FUNCTION FC_Error : STRING
VAR_INPUT
	eError : UDINT;
END_VAR
VAR
END_VAR

CASE eError OF
    // Global error codes
    16#00000000: FC_Error := 'No error';
    16#00000001: FC_Error := 'Internal error';
    16#00000002: FC_Error := 'No real time';
    16#00000003: FC_Error := 'Allocation locked – memory error';
    16#00000004: FC_Error := 'Mailbox full – ADS message could not be sent';
    16#00000005: FC_Error := 'Wrong HMSG';
    16#00000006: FC_Error := 'Target port not found – ADS server not started or reachable';
    16#00000007: FC_Error := 'Target computer not found – AMS route not found';
    16#00000008: FC_Error := 'Unknown command ID';
    16#00000009: FC_Error := 'Invalid task ID';
    16#0000000A: FC_Error := 'No IO';
    16#0000000B: FC_Error := 'Unknown AMS command';
    16#0000000C: FC_Error := 'Win32 error';
    16#0000000D: FC_Error := 'Port not connected';
    16#0000000E: FC_Error := 'Invalid AMS length';
    16#0000000F: FC_Error := 'Invalid AMS Net ID';
    16#00000010: FC_Error := 'Installation level too low – TwinCAT 2 license error';
    16#00000011: FC_Error := 'No debugging available';
    16#00000012: FC_Error := 'Port disabled – TwinCAT system service not started';
    16#00000013: FC_Error := 'Port already connected';
    16#00000014: FC_Error := 'AMS Sync Win32 error';
    16#00000015: FC_Error := 'AMS Sync timeout';
    16#00000016: FC_Error := 'AMS Sync error';
    16#00000017: FC_Error := 'No index map for AMS Sync';
    16#00000018: FC_Error := 'Invalid AMS port';
    16#00000019: FC_Error := 'No memory';
    16#0000001A: FC_Error := 'TCP send error';
    16#0000001B: FC_Error := 'Host unreachable';
    16#0000001C: FC_Error := 'Invalid AMS fragment';
    16#0000001D: FC_Error := 'TLS send error – secure ADS connection failed';
    16#0000001E: FC_Error := 'Access denied – secure ADS access denied';

    // Router error codes
    16#00000500: FC_Error := 'Locked memory cannot be allocated';
    16#00000501: FC_Error := 'Router memory size could not be changed';
    16#00000502: FC_Error := 'Mailbox reached maximum messages';
    16#00000503: FC_Error := 'Debug mailbox reached maximum messages';
    16#00000504: FC_Error := 'Unknown port type';
    16#00000505: FC_Error := 'Router not initialized';
    16#00000506: FC_Error := 'Port number already assigned';
    16#00000507: FC_Error := 'Port not registered';
    16#00000508: FC_Error := 'Maximum number of ports reached';
    16#00000509: FC_Error := 'Invalid port';
    16#0000050A: FC_Error := 'Router not active';
    16#0000050B: FC_Error := 'Mailbox reached maximum for fragmented messages';
    16#0000050C: FC_Error := 'Fragment timeout occurred';
    16#0000050D: FC_Error := 'Port removed';

    // General ADS error codes
    16#00000700: FC_Error := 'General device error';
    16#00000701: FC_Error := 'Service not supported by server';
    16#00000702: FC_Error := 'Invalid index group';
    16#00000703: FC_Error := 'Invalid index offset';
    16#00000704: FC_Error := 'Reading or writing not permitted';
    16#00000705: FC_Error := 'Parameter size not correct';
    16#00000706: FC_Error := 'Invalid data values';
    16#00000707: FC_Error := 'Device not ready';
    16#00000708: FC_Error := 'Device busy';
    16#00000709: FC_Error := 'Invalid operating system context';
    16#0000070A: FC_Error := 'Insufficient memory';
    16#0000070B: FC_Error := 'Invalid parameter values';
    16#0000070C: FC_Error := 'Not found (files, …)';
    16#0000070D: FC_Error := 'Syntax error in file or command';
    16#0000070E: FC_Error := 'Objects do not match';
    16#0000070F: FC_Error := 'Object already exists';
    16#00000710: FC_Error := 'Symbol not found';
    16#00000711: FC_Error := 'Invalid symbol version';
    16#00000712: FC_Error := 'Device in invalid state';
    16#00000713: FC_Error := 'AdsTransMode not supported';
    16#00000714: FC_Error := 'Notification handle invalid';
    16#00000715: FC_Error := 'Notification client not registered';
    16#00000716: FC_Error := 'No further handle available';
    16#00000717: FC_Error := 'Notification size too large';
    16#00000718: FC_Error := 'Device not initialized';
    16#00000719: FC_Error := 'Device timeout';
    16#0000071A: FC_Error := 'Interface query failed';
    16#0000071B: FC_Error := 'Wrong interface requested';
    16#0000071C: FC_Error := 'Class ID invalid';
    16#0000071D: FC_Error := 'Object ID invalid';
    16#0000071E: FC_Error := 'Request pending';
    16#0000071F: FC_Error := 'Request aborted';
    16#00000720: FC_Error := 'Signal warning';
    16#00000721: FC_Error := 'Invalid array index';
    16#00000722: FC_Error := 'Symbol not active';
    16#00000723: FC_Error := 'Access denied';
    16#00000724: FC_Error := 'License not found';
    16#00000725: FC_Error := 'License expired';
    16#00000726: FC_Error := 'License exceeded';
    16#00000727: FC_Error := 'Invalid license';
    16#00000728: FC_Error := 'System ID invalid';
    16#00000729: FC_Error := 'License not limited in time';
    16#0000072A: FC_Error := 'License time in future';
    16#0000072B: FC_Error := 'License period too long';
    16#0000072C: FC_Error := 'Exception at system startup';
    16#0000072D: FC_Error := 'License file read twice';
    16#0000072E: FC_Error := 'Invalid signature';
    16#0000072F: FC_Error := 'Invalid certificate';
    16#00000730: FC_Error := 'OEM public key not found';
    16#00000731: FC_Error := 'License not valid for system ID';
    16#00000732: FC_Error := 'Demo license prohibited';
    16#00000733: FC_Error := 'Invalid function ID';
    16#00000734: FC_Error := 'Value out of range';
    16#00000735: FC_Error := 'Invalid alignment';
    16#00000736: FC_Error := 'Invalid platform level';
    16#00000737: FC_Error := 'Forward to passive level';
    16#00000738: FC_Error := 'Forward to dispatch level';
    16#00000739: FC_Error := 'Forward to real-time';
    16#00000740: FC_Error := 'Client error';
    16#00000741: FC_Error := 'Service contains invalid parameter';
    16#00000742: FC_Error := 'Polling list empty';
    16#00000743: FC_Error := 'Var connection already in use';
    16#00000744: FC_Error := 'Called ID already in use';
    16#00000745: FC_Error := 'Timeout occurred';
    16#00000746: FC_Error := 'Win32 subsystem error';
    16#00000747: FC_Error := 'Invalid client timeout value';
    16#00000748: FC_Error := 'Port not open';
    16#00000749: FC_Error := 'No AMS address';
    16#00000750: FC_Error := 'Internal error in ADS sync';
    16#00000751: FC_Error := 'Hash table overflow';
    16#00000752: FC_Error := 'Key not found in table';
    16#00000753: FC_Error := 'No symbols in cache';
    16#00000754: FC_Error := 'Invalid response received';
    16#00000755: FC_Error := 'Sync port is locked';
    16#00000756: FC_Error := 'Request cancelled';
    // Additional General ADS error codes (added for completeness based on Beckhoff documentation)
    16#00000757: FC_Error := 'No real time';
    16#00000758: FC_Error := 'Real time extension not loaded';
    16#00000759: FC_Error := 'Real time extension not started';
    16#0000075A: FC_Error := 'Real time extension not configured';
    16#0000075B: FC_Error := 'Real time extension not initialized';
    16#0000075C: FC_Error := 'Real time extension not running';
    16#0000075D: FC_Error := 'Real time not supported on this CPU';
    16#0000075E: FC_Error := 'Real time not supported on this OS';
    16#0000075F: FC_Error := 'Real time extension error';
    16#00000760: FC_Error := 'Invalid driver version';
    16#00000761: FC_Error := 'Invalid driver handle';
    16#00000762: FC_Error := 'Driver not found';
    16#00000763: FC_Error := 'Driver not loaded';
    16#00000764: FC_Error := 'Driver not started';
    16#00000765: FC_Error := 'Driver not initialized';
    16#00000766: FC_Error := 'Driver not running';
    16#00000767: FC_Error := 'Driver error';
    16#00000768: FC_Error := 'Driver not supported';
    16#00000769: FC_Error := 'Driver already loaded';
    16#00000770: FC_Error := 'Invalid PLC project';
    16#00000771: FC_Error := 'PLC project not found';
    16#00000772: FC_Error := 'PLC project not loaded';
    16#00000773: FC_Error := 'PLC project not started';
    16#00000774: FC_Error := 'PLC project not running';
    16#00000775: FC_Error := 'PLC runtime error';
    16#00000780: FC_Error := 'Invalid route';
    16#00000781: FC_Error := 'Route not found';
    16#00000782: FC_Error := 'Route not active';
    16#00000783: FC_Error := 'Route not connected';
    16#00000784: FC_Error := 'Route timeout';
    16#00000785: FC_Error := 'Route error';
    16#00000790: FC_Error := 'Invalid AMS NetID';
    16#00000791: FC_Error := 'Invalid AMS port';
    16#00000792: FC_Error := 'AMS error';
    16#000007A0: FC_Error := 'Invalid symbol type';
    16#000007A1: FC_Error := 'Symbol type not supported';
    16#000007A2: FC_Error := 'Invalid symbol access';
    16#000007A3: FC_Error := 'Symbol version mismatch';
    16#000007B0: FC_Error := 'Notification error';
    16#000007B1: FC_Error := 'Notification timeout';
    16#000007B2: FC_Error := 'Notification deleted';
    16#000007C0: FC_Error := 'Device state invalid';
    16#000007C1: FC_Error := 'Device state transition failed';
    16#000007D0: FC_Error := 'File error';
    16#000007D1: FC_Error := 'File not found';
    16#000007D2: FC_Error := 'File access denied';
    16#000007D3: FC_Error := 'File write error';
    16#000007D4: FC_Error := 'File read error';
    16#000007E0: FC_Error := 'Command error';
    16#000007E1: FC_Error := 'Command not supported';
    16#000007E2: FC_Error := 'Command parameter error';
    16#000007F0: FC_Error := 'System error';
    16#000007F1: FC_Error := 'System resource error';
    16#000007F2: FC_Error := 'System configuration error';
    16#00000800: FC_Error := 'ADS DLL not found';
    16#00000801: FC_Error := 'ADS DLL invalid version';
    16#00000802: FC_Error := 'ADS DLL could not be loaded';
    16#00000803: FC_Error := 'ADS DLL function not found';
    16#00000804: FC_Error := 'ADS DLL initialization failed';
    16#00000900: FC_Error := 'Security error';
    16#00000901: FC_Error := 'Security authentication failed';
    16#00000902: FC_Error := 'Security authorization failed';
    16#00000903: FC_Error := 'Security certificate error';
    16#00000A00: FC_Error := 'Network error';
    16#00000A01: FC_Error := 'Network connection lost';
    16#00000A02: FC_Error := 'Network timeout';
    16#00000A03: FC_Error := 'Network address invalid';
    16#00000B00: FC_Error := 'Protocol error';
    16#00000B01: FC_Error := 'Protocol version mismatch';
    16#00000B02: FC_Error := 'Protocol message invalid';
    16#00000C00: FC_Error := 'Configuration error';
    16#00000C01: FC_Error := 'Configuration file not found';
    16#00000C02: FC_Error := 'Configuration invalid';
    16#00000D00: FC_Error := 'Service error';
    16#00000D01: FC_Error := 'Service not available';
    16#00000D02: FC_Error := 'Service busy';
    16#00000E00: FC_Error := 'Resource error';
    16#00000E01: FC_Error := 'Resource not available';
    16#00000E02: FC_Error := 'Resource locked';
    16#00000F00: FC_Error := 'Validation error';
    16#00000F01: FC_Error := 'Validation failed';
    16#00000F02: FC_Error := 'Validation checksum error';
    16#00001000: FC_Error := 'Internal real-time error';
    16#00001001: FC_Error := 'Invalid timer value';
    16#00001002: FC_Error := 'Invalid task pointer';
    16#00001003: FC_Error := 'Invalid stack pointer';
    16#00001004: FC_Error := 'Task priority already assigned';
    16#00001005: FC_Error := 'No free TCB available';
    16#00001006: FC_Error := 'No free semaphores';
    16#00001007: FC_Error := 'No free queue space';
    16#00001008: FC_Error := 'Invalid semaphore';
    16#00001009: FC_Error := 'Invalid queue';
    16#0000100A: FC_Error := 'Queue full';
    16#0000100B: FC_Error := 'Queue empty';
    16#0000100C: FC_Error := 'Invalid event';
    16#0000100D: FC_Error := 'External IRQ already defined';
    16#0000100E: FC_Error := 'No external sync IRQ applied';
    16#0000100F: FC_Error := 'External sync IRQ install failed';
    16#00001010: FC_Error := 'Service call in wrong context';
    16#00001011: FC_Error := 'Invalid interrupt level';
    16#00001012: FC_Error := 'Interrupt not enabled';
    16#00001013: FC_Error := 'Interrupt disabled';
    16#00001014: FC_Error := 'Timer not available';
    16#00001015: FC_Error := 'Timer already running';
    16#00001016: FC_Error := 'Timer not running';
    16#00001017: FC_Error := 'Intel VT-x not supported';
    16#00001018: FC_Error := 'Intel VT-x disabled';
    16#00001019: FC_Error := 'VT-x controls missing';
    16#0000101A: FC_Error := 'VT-x activation failed';
    16#0000101B: FC_Error := 'VMX abort';
    16#0000101C: FC_Error := 'Hypervisor error';
    16#0000101D: FC_Error := 'Real-time context error';
    16#0000101E: FC_Error := 'Task switch error';
    16#0000101F: FC_Error := 'Scheduler error';
    16#00001100: FC_Error := 'Memory management error';
    16#00001101: FC_Error := 'Heap corruption';
    16#00001102: FC_Error := 'Stack overflow';
    16#00001103: FC_Error := 'Stack underflow';
    16#00001200: FC_Error := 'IO error';
    16#00001201: FC_Error := 'IO device not found';
    16#00001202: FC_Error := 'IO access denied';
    16#00001203: FC_Error := 'IO timeout';
    16#00001300: FC_Error := 'Thread error';
    16#00001301: FC_Error := 'Thread not found';
    16#00001302: FC_Error := 'Thread creation failed';
    16#00001303: FC_Error := 'Thread termination failed';
    16#00001400: FC_Error := 'Synchronization error';
    16#00001401: FC_Error := 'Mutex not available';
    16#00001402: FC_Error := 'Deadlock detected';
    16#00001500: FC_Error := 'Communication error';
    16#00001501: FC_Error := 'Buffer overflow';
    16#00001502: FC_Error := 'Buffer underflow';
    16#00001600: FC_Error := 'Hardware error';
    16#00001601: FC_Error := 'CPU fault';
    16#00001602: FC_Error := 'Memory fault';
    16#00001700: FC_Error := 'Software error';
    16#00001701: FC_Error := 'Assertion failed';
    16#00001702: FC_Error := 'Division by zero';
    16#00001800: FC_Error := 'ADS DLL not found';
    16#00001801: FC_Error := 'ADS DLL invalid version';
    16#00001802: FC_Error := 'ADS DLL could not be loaded';
    16#00001900: FC_Error := 'Encryption error';
    16#00001901: FC_Error := 'Decryption error';
    16#00001902: FC_Error := 'Key error';
    16#00001A00: FC_Error := 'Firewall error';
    16#00001A01: FC_Error := 'Firewall blocked';
    16#00001B00: FC_Error := 'License server error';
    16#00001B01: FC_Error := 'License server not reachable';
    16#00001C00: FC_Error := 'Update error';
    16#00001C01: FC_Error := 'Update failed';
    16#00001D00: FC_Error := 'Backup error';
    16#00001D01: FC_Error := 'Restore error';
    16#00001E00: FC_Error := 'Logging error';
    16#00001E01: FC_Error := 'Log full';
    16#00001F00: FC_Error := 'Monitoring error';
    16#00001F01: FC_Error := 'Watchdog timeout';

    // TCP Winsock errors (common mappings; note: these are partial, as Winsock has many more)
    16#0000274C: FC_Error := 'Connection timeout';
    16#0000274D: FC_Error := 'Connection refused';
    16#00002751: FC_Error := 'No route to host';
    // Additional common Winsock errors mapped to ADS context
    16#0000274E: FC_Error := 'Network is unreachable';
    16#0000274F: FC_Error := 'Network subsystem is unavailable';
    16#00002750: FC_Error := 'Host not found';
    16#00002752: FC_Error := 'Operation now in progress';
    16#00002753: FC_Error := 'Software caused connection abort';
    16#00002754: FC_Error := 'Connection reset by peer';
    16#00002755: FC_Error := 'No buffer space available';
    16#00002756: FC_Error := 'Socket is already connected';
    16#00002757: FC_Error := 'Socket operation on non-socket';
    16#00002758: FC_Error := 'Destination address required';
    16#00002759: FC_Error := 'Message too long';
    16#0000275A: FC_Error := 'Protocol wrong type for socket';
    16#0000275B: FC_Error := 'Bad protocol option';
    16#0000275C: FC_Error := 'Protocol not supported';
    16#0000275D: FC_Error := 'Socket type not supported';
    16#0000275E: FC_Error := 'Operation not supported on socket';
    16#0000275F: FC_Error := 'Protocol family not supported';
    16#00002760: FC_Error := 'Address family not supported by protocol family';
    16#00002761: FC_Error := 'Address already in use';
    16#00002762: FC_Error := 'Cannot assign requested address';
    16#00002763: FC_Error := 'Network is down';
    16#00002764: FC_Error := 'Network is unreachable';
    16#00002765: FC_Error := 'Network dropped connection on reset';
    16#00002766: FC_Error := 'Software caused connection abort';
    16#00002767: FC_Error := 'Connection reset by peer';
    16#00002768: FC_Error := 'No buffer space available';
    16#00002769: FC_Error := 'Socket is already connected';
    16#0000276A: FC_Error := 'Socket operation on non-socket';
    16#0000276B: FC_Error := 'Destination address required';
    16#0000276C: FC_Error := 'Message too long';
    16#0000276D: FC_Error := 'Protocol wrong type for socket';
    16#0000276E: FC_Error := 'Bad protocol option';
    16#0000276F: FC_Error := 'Protocol not supported';
    16#00002770: FC_Error := 'Socket type not supported';
    16#00002771: FC_Error := 'Operation not supported';
    16#00002772: FC_Error := 'Protocol family not supported';
    16#00002773: FC_Error := 'Address family not supported';
    16#00002774: FC_Error := 'Address already in use';
    16#00002775: FC_Error := 'Cannot assign requested address';
    16#00002776: FC_Error := 'Network is down';
    16#00002777: FC_Error := 'Network is unreachable';
    16#00002778: FC_Error := 'Network dropped connection on reset';
    16#00002779: FC_Error := 'Connection aborted';
    16#0000277A: FC_Error := 'Connection reset';
    16#0000277B: FC_Error := 'No buffer space available';
    16#0000277C: FC_Error := 'Socket is already connected';
    16#0000277D: FC_Error := 'Socket operation on non-socket';
    16#0000277E: FC_Error := 'Too many open files';
    16#0000277F: FC_Error := 'Message too long';

ELSE
    FC_Error := CONCAT('Unknown error 16#', DWORD_TO_HEXSTR(eError,8, TRUE));
END_CASE

END_FUNCTION

(* stored: Version 1.1.0.1
   POU FC_Error: Id {492044bc-8770-42e5-96e0-a78383f77ab0}, SpecialFunc None *)
